FUNCTION_BLOCK fb_io_in_bool
VAR_INPUT
	hw_value AT %I* 	: BOOL;
	SimFlag:BOOL;
	SimValue:BOOL:=TRUE;
END_VAR
VAR_OUTPUT
	Value:BOOL;
END_VAR
VAR
END_VAR


IF SimFlag THEN
	Value:= SimValue;
ELSE
	value:= hw_value;
END_IF

END_FUNCTION_BLOCK

(* stored: Version 1.1.0.1, ProductVersion 3.1.4024.3
   POU fb_io_in_bool: Id {cb366695-a736-429b-8ba9-a477ce532cee}, SpecialFunc None *)
